{attribute 'hide_all_locals'}
FUNCTION_BLOCK FB_MotionSyncPrivate
VAR_INPUT
END_VAR
VAR_OUTPUT
END_VAR
VAR
    // private vars for data exchange
    eSynPrvAxisState : MC_AxisStates;
    bSynPrvReset : BOOL;
    bSynPrvEnable :BOOL;
    bSynPrvPowerEn : BOOL;
    bSynPrvExec : BOOL;
    bSynPrvError : BOOL;
    bSynPrvHomeBusy : BOOL;
    bSynPrvLocalExec : BOOL;
    bSynPrvLimHit : BOOL := TRUE;
    bSynPrvMoveBusy : BOOL;
    bSynPrvMoveDone : BOOL;
    bSynPrvNewMoveReq : BOOL;
    bSynPrvAllFwdEn: BOOL:=FALSE;
    bSynPrvAllBwdEn: BOOL:=FALSE;
    bSynPrvAllEn: BOOL:=FALSE;
    bSynPrvLimFwd : BOOL:=FALSE;
    bSynPrvLimBwd : BOOL:=FALSE;
    bSynPrvHome: BOOL:=TRUE;
END_VAR

PROPERTY RestoreDone : BOOL
GET
END_GET
SET
END_SET
END_PROPERTY

PROPERTY INTERNAL SynPrvAllBwdEn : BOOL
GET
SynPrvAllBwdEn := bSynPrvAllBwdEn;
END_GET
SET
bSynPrvAllBwdEn := SynPrvAllBwdEn;
END_SET
END_PROPERTY

PROPERTY INTERNAL SynPrvAllEn : BOOL
GET
SynPrvAllEn := bSynPrvAllEn;
END_GET
SET
bSynPrvAllEn := SynPrvAllEn;
END_SET
END_PROPERTY

PROPERTY INTERNAL SynPrvAllFwdEn : BOOL
GET
SynPrvAllFwdEn := bSynPrvAllFwdEn;
END_GET
SET
bSynPrvAllFwdEn := SynPrvAllFwdEn;
END_SET
END_PROPERTY

PROPERTY INTERNAL SynPrvAxisState : MC_AxisStates
GET
SynPrvAxisState := eSynPrvAxisState;
END_GET
SET
eSynPrvAxisState := SynPrvAxisState;
END_SET
END_PROPERTY

PROPERTY INTERNAL SynPrvError : BOOL
GET
SynPrvError := bSynPrvError;
END_GET
SET
bSynPrvError := SynPrvError;
END_SET
END_PROPERTY

PROPERTY INTERNAL SynPrvExec : BOOL
GET
SynPrvExec := bSynPrvExec;
END_GET
SET
bSynPrvExec := SynPrvExec;
END_SET
END_PROPERTY

PROPERTY INTERNAL SynPrvHome : BOOL
GET
SynPrvHome := bSynPrvHome;
END_GET
SET
bSynPrvHome := SynPrvHome;
END_SET
END_PROPERTY

PROPERTY INTERNAL SynPrvHomeBusy : BOOL
GET
SynPrvHomeBusy := bSynPrvHomeBusy ;
END_GET
SET
bSynPrvHomeBusy := SynPrvHomeBusy;
END_SET
END_PROPERTY

PROPERTY INTERNAL SynPrvLimBwd : BOOL
GET
SynPrvLimBwd := bSynPrvLimBwd;
END_GET
SET
END_SET
END_PROPERTY

PROPERTY INTERNAL SynPrvLimFwd : BOOL
GET
SynPrvLimFwd := bSynPrvLimFwd;
END_GET
SET
bSynPrvLimFwd := SynPrvLimFwd;
END_SET
END_PROPERTY

PROPERTY INTERNAL SynPrvLimHit : BOOL
GET
SynPrvLimHit := bSynPrvLimHit;
END_GET
SET
bSynPrvLimHit :=SynPrvLimHit;
END_SET
END_PROPERTY

PROPERTY INTERNAL SynPrvLocalExec : BOOL
GET
SynPrvLocalExec := bSynPrvLocalExec;
END_GET
SET
bSynPrvLocalExec := SynPrvLocalExec;
END_SET
END_PROPERTY

PROPERTY INTERNAL SynPrvMoveBusy : BOOL
GET
SynPrvMoveBusy := bSynPrvMoveBusy;
END_GET
SET
bSynPrvMoveBusy := SynPrvMoveBusy;
END_SET
END_PROPERTY

PROPERTY INTERNAL SynPrvMoveDone : BOOL
GET
SynPrvMoveDone := bSynPrvMoveDone;
END_GET
SET
bSynPrvMoveDone := SynPrvMoveDone;
END_SET
END_PROPERTY

PROPERTY INTERNAL SynPrvNewMoveReq : BOOL
GET
SynPrvNewMoveReq := bSynPrvNewMoveReq;
END_GET
SET
bSynPrvNewMoveReq := SynPrvNewMoveReq;
END_SET
END_PROPERTY

PROPERTY INTERNAL SynPrvPowerEn : BOOL
GET
SynPrvPowerEn := bSynPrvPowerEn;
END_GET
SET
bSynPrvPowerEn := SynPrvPowerEn;
END_SET
END_PROPERTY

PROPERTY INTERNAL SynPrvReset : BOOL
GET
SynPrvReset := bSynPrvReset;
END_GET
SET
bSynPrvReset := SynPrvReset;
END_SET
END_PROPERTY

END_FUNCTION_BLOCK

(* stored: Version 1.1.0.1
   POU FB_MotionSyncPrivate: Id {c8657e3e-5d0e-4fad-8966-c25217ba52eb}, SpecialFunc None
   Property RestoreDone: Id {bf833be0-1689-4371-bd70-cc4a0bf77765}
   Get Get: Id {a6680489-5f82-4020-876d-3a889009fbc1}
   Set Set: Id {72546998-d228-4251-9151-7bb114efff40}
   Property SynPrvAllBwdEn: Id {f6d0f8df-5d1b-4ff4-8d72-c759807caf80}
   Get Get: Id {adc014ce-aa13-4a87-97fb-07539f9d4700}
   Set Set: Id {380e996d-7248-4d33-8d3f-65fb41575fda}
   Property SynPrvAllEn: Id {c0de1886-8603-49b1-a42c-e1d3245d918a}
   Get Get: Id {af6eba22-2060-4acb-8932-1f88130efba2}
   Set Set: Id {70ff85b4-8da3-4e54-a370-45e963a0717e}
   Property SynPrvAllFwdEn: Id {196240ef-5413-416d-b0a0-36403e6a22fd}
   Get Get: Id {eb353156-a9c5-4bf9-9328-925ec78072c1}
   Set Set: Id {22e1b304-704e-415e-9f83-894f4cbecebf}
   Property SynPrvAxisState: Id {60919b8b-a0ee-4b61-b888-5912d190160f}
   Get Get: Id {2a6fc420-bce2-4a3d-b8e7-0fc168de1ca2}
   Set Set: Id {78296327-b508-4ee5-b38e-cefa436e41c3}
   Property SynPrvError: Id {1b6034c0-b26d-469a-a57b-82a6b4ebb40e}
   Get Get: Id {2090a12b-697a-474d-8f07-02cf7adb2cfa}
   Set Set: Id {92c801ed-d007-4f8d-9ca0-37d8d73043c4}
   Property SynPrvExec: Id {f59250e2-9c98-4c00-b85c-b271e1e66ae9}
   Get Get: Id {889b001c-f145-4973-a9c8-4b26c4b13927}
   Set Set: Id {415a2309-d0bb-4d9a-be5d-8503058c5b92}
   Property SynPrvHome: Id {4a596f7b-8cd3-4101-8575-8cf898fbea0e}
   Get Get: Id {b38e456d-0618-424d-b236-77052140716c}
   Set Set: Id {af0ee15c-32ca-4568-9855-6b4fa1b56389}
   Property SynPrvHomeBusy: Id {4dbef2a8-0478-4d7e-8785-7f84f70fd518}
   Get Get: Id {bad28b9c-c267-4ef7-af8c-55a86c0b0457}
   Set Set: Id {513660d9-a9bd-4d34-a48c-2fbb590949d5}
   Property SynPrvLimBwd: Id {f32a3277-e991-4dbe-b8fd-3c81a0c59dfc}
   Get Get: Id {7473e81f-bbcc-4d89-a8c1-2765010f18e7}
   Set Set: Id {baf2e00b-623d-4734-af90-c7149b700472}
   Property SynPrvLimFwd: Id {12a0e278-6936-49c1-85f0-c147c4f8d84a}
   Get Get: Id {754501d6-96ab-4a3f-bc61-40e52ad936a5}
   Set Set: Id {91808e78-aeef-4059-9a0d-b2a046ceed2c}
   Property SynPrvLimHit: Id {48dba4e9-594a-4aa6-8b94-cff3ad033b6c}
   Get Get: Id {583b7193-cfed-4323-b867-2c22006efc55}
   Set Set: Id {7fed7d13-1613-4f0a-95ad-773f423ee6e8}
   Property SynPrvLocalExec: Id {55e60caf-15fb-484d-be9e-bfc64626c188}
   Get Get: Id {c56dd8e1-9f86-464e-9efe-ae4518446f87}
   Set Set: Id {526b5cf7-cfa7-4416-ad4d-9435459172c6}
   Property SynPrvMoveBusy: Id {15420f33-1dbf-440d-ad57-611e93f2e318}
   Get Get: Id {702d2cf3-0c44-4bac-b8a8-197105c16a79}
   Set Set: Id {91e71f84-421a-40b0-8aee-098563bc8eba}
   Property SynPrvMoveDone: Id {48b7baf8-ed4e-4bb9-847e-f1327eadbca1}
   Get Get: Id {55f2c259-1d28-4c69-9ed3-51bd0af0ee15}
   Set Set: Id {96610def-86e6-4cbb-8e04-79b3050eaba1}
   Property SynPrvNewMoveReq: Id {99d1eaeb-20b7-470e-97ca-8e71ab6dc340}
   Get Get: Id {b91286bc-c75d-4cbe-81e2-ebc4d5686439}
   Set Set: Id {dd931d0f-9513-4185-a887-4ff73f9de3a8}
   Property SynPrvPowerEn: Id {b485bb6e-31db-4da3-a959-a64f2de8176d}
   Get Get: Id {ac508b0b-6085-4d54-ba10-918184705e91}
   Set Set: Id {273113d6-170f-4eaf-8a28-b9222afd00a2}
   Property SynPrvReset: Id {115cac90-f6aa-4f95-a966-8d415f1cee88}
   Get Get: Id {e76d1538-b8db-4fd9-9610-382e5e0fc2f5}
   Set Set: Id {fa3aab3c-f3be-4f32-a557-a380bd9b85c0} *)
